(* PLC project Anjlab Code Box, Prosoft-Systems Ltd. Astra.IDE Astra.IDE_V1.7.2.1, author Sergey A Glukhov *)
(* stored: creationDateTime 2025-06-12T14:05:23.9971404, version 3.5.17.1, modificationDateTime 2025-06-12T13:59:54.8513333, organization Anjlab *)
(* Helpful ST blocks and functions *)

(* Сглаживание дискретного сигнала *)
FUNCTION_BLOCK DebunceBoolIn
  VAR_INPUT
    input : BOOL;  (* Входной сигнал *)
  END_VAR
  VAR_OUTPUT
    output : BOOL;  (* Выходной сигнал *)
  END_VAR
  VAR
    startTime : TIME;  (* Время начала *)
    memory : BOOL;  (* Память сигнала *)
  END_VAR

            IF input AND NOT memory THEN
	startTime := TIME();
END_IF;
memory := input;
output := input AND ((TIME() - startTime) > T#100ms);
          
END_FUNCTION_BLOCK

(* Сглаживание дискретного сигнала *)
FUNCTION_BLOCK DebunceBoolInOut
  VAR_INPUT
    input : BOOL;  (* Входной сигнал *)
  END_VAR
  VAR_OUTPUT
    output : BOOL;  (* Выходной сигнал *)
  END_VAR
  VAR
    startTime : TIME;  (* Время начала *)
    memory : BOOL;  (* Память сигнала *)
  END_VAR

            IF (NOT input AND memory) OR (input AND NOT memory) THEN
	startTime := TIME();
END_IF;
memory := input;
output := input;
IF ((TIME() - startTime) < T#100ms) THEN
	output := NOT input;
END_IF
          
END_FUNCTION_BLOCK

(* Сглаживание дискретного сигнала *)
FUNCTION_BLOCK DebunceBoolOut
  VAR_INPUT
    input : BOOL;  (* Входной сигнал *)
  END_VAR
  VAR_OUTPUT
    output : BOOL;  (* Выходной сигнал *)
  END_VAR
  VAR
    startTime : TIME;  (* Время начала *)
    memory : BOOL;  (* Память сигнала *)
  END_VAR

            IF NOT input AND memory THEN
	startTime := TIME();
END_IF;
memory := input;
output := input;
IF NOT input AND ((TIME() - startTime) < T#100ms) THEN
	output := TRUE;
END_IF
          
END_FUNCTION_BLOCK

(* выделяет передний и задний фронт с фильтром на 100 миллисекунд *)
FUNCTION_BLOCK DetectEdgeFiltered
  VAR_INPUT
    input : BOOL;  (* Входной сигнал *)
  END_VAR
  VAR_OUTPUT
    raise : BOOL;  (* Передний фронт *)
    fall : BOOL;  (* Задний фронт *)
  END_VAR
  VAR
    fbDio1 : DebunceBoolInOut;
    filteredInput : BOOL;  (* Отфильтрованный вход *)
    memory : BOOL;
  END_VAR

            fbDio1(input := input, output => filteredInput);
raise := fall := FALSE;
IF filteredInput AND NOT memory THEN
	raise := TRUE;
ELSIF NOT filteredInput AND memory THEN
	fall := TRUE;
END_IF
memory := filteredInput;
          
END_FUNCTION_BLOCK

(* Двойной клик *)
FUNCTION_BLOCK DoubleClick
  VAR_INPUT
    input : BOOL;  (* Входной сигнал *)
  END_VAR
  VAR_OUTPUT
    output : BOOL;  (* Выходной сигнал *)
  END_VAR
  VAR
    startTime : TIME;  (* Время начала *)
    memory : BOOL;  (* Память сигнала *)
  END_VAR

            output := FALSE;
IF input AND NOT memory THEN
	IF (TIME() - startTime) > T#100MS AND (TIME() - startTime) < T#800MS THEN
		output := TRUE;
	END_IF;
	startTime := TIME();
END_IF;
memory := input;
          
END_FUNCTION_BLOCK

(* Эта функция хранит до 32-х значений в буфере и выдает среднее значение. Вы сами можете решить, сколько значений сохранить для получения среднего числа. *)
FUNCTION_BLOCK FilterNR
  VAR_INPUT
    input : WORD;  (* Входное значение *)
    bufferSize : UINT;  (* Размер буфера минимум 32 максимум 1000 *)
    reset : BOOL;  (* Сброс буфера *)
  END_VAR
  VAR_OUTPUT
    output : WORD;  (* Выходное отфильтрованное значение *)
  END_VAR
  VAR
    isInitialized : BOOL;
    buffer : ARRAY[1..1000] OF WORD;
    counter : UINT;
    sum : DINT;
  END_VAR

            (* ограничим bufferSize в размер буфера *)
bufferSize := MIN(MAX(bufferSize, 1000), 32);
(* Инициализация *)
IF NOT isInitialized OR reset THEN
	isInitialized := TRUE;
	FOR counter := 1 TO bufferSize DO
		buffer[counter] := input;
	END_FOR;
	sum := input * bufferSize;
	output := input;
	RETURN;
END_IF;

IF counter >= bufferSize THEN
    counter := 1;
ELSE
    counter := counter + 1;
END_IF

sum := sum + input - buffer[counter];
{warning disable C0195}
output := DWORD_TO_WORD(sum / bufferSize);
buffer[counter] := input;
          
END_FUNCTION_BLOCK

(* возвращает среднее значение за определенный промежуток времени. *)
FUNCTION_BLOCK FilterTW
  VAR_INPUT
    input : WORD;  (* Входное значение *)
    timeInterval : TIME;  (* Временной интервал *)
  END_VAR
  VAR_OUTPUT
    output : WORD;  (* Выходное отфильтрованное значение *)
  END_VAR
  VAR
    isInitialized : BOOL;
    currentTime : DWORD;
    lastTime : DWORD;
    tempTime : DWORD;
  END_VAR

            (* Получаем текущее время *)
currentTime := TIME_TO_DWORD(TIME());
(* Инициализация *)
IF NOT isInitialized OR timeInterval = T#0s THEN
	isInitialized := TRUE;
	lastTime := currentTime;
	output := input;
ELSIF output = input THEN
	lastTime := currentTime;
ELSE
	tempTime := WORD_TO_DWORD(input - output) * (currentTime - lastTime) /
	TIME_TO_DWORD(timeInterval);
	IF tempTime <> 0 THEN
		output := DINT_TO_WORD(WORD_TO_DINT(output) + DWORD_TO_DINT(tempTime));
		lastTime := currentTime;
	END_IF;
END_IF;
          
END_FUNCTION_BLOCK

(* Долгий клик *)
FUNCTION_BLOCK LongClick
  VAR_INPUT
    input : BOOL;  (* Входной сигнал *)
    pressTime : TIME;  (* Время нажатия *)
  END_VAR
  VAR_OUTPUT
    output : BOOL;  (* Выходной сигнал *)
  END_VAR
  VAR
    startTime : TIME;  (* Время начала *)
    memory : BOOL;  (* Память сигнала *)
  END_VAR

            IF input AND NOT memory THEN
	startTime := TIME();
END_IF;
memory := input;
output := input AND ((TIME() - startTime) > pressTime);
          
END_FUNCTION_BLOCK

(* создает импульсы с заданной частотой CLK_PWM(EN := TRUE, PT := T#5ms); На выходе Q будет импульс в один цикл ПЛК, раз в 5 миллисекунд. *)
FUNCTION_BLOCK PwmClock
  VAR_INPUT
    enable : BOOL;  (* Запуск генератора *)
    pulseTime : TIME := TIME#10ms;  (* Время импульсов *)
  END_VAR
  VAR_OUTPUT
    output : BOOL;  (* Выходной сигнал *)
  END_VAR
  VAR
    memory : BOOL;
    lastTime : TIME;
    currentTime : TIME;
  END_VAR

            currentTime := TIME();
IF enable AND NOT memory THEN
	lastTime := currentTime - pulseTime;
END_IF;
memory := enable;
output := currentTime - lastTime >= pulseTime;
IF output THEN lastTime := currentTime; END_IF;
          
END_FUNCTION_BLOCK

(* создает ШИМ-сигнал заданной частоты со смещением соотношения. Каждый цик ШИМ можно разделить на 2 фазы: Ton (время включения) и Toff (время выключения). Соотношение задается от 0 до 1. Например, соотношение 0.5 разделит время каждого цикла шим на 50% на Ton и 50% на Toff . *)
FUNCTION_BLOCK PwmDc
  VAR_INPUT
    frequency : REAL;  (* Частота, раз в секунду (Гц) *)
    dutyCycle : REAL;  (* Соотношение *)
  END_VAR
  VAR_OUTPUT
    output : BOOL;  (* Выходной сигнал *)
  END_VAR
  VAR
    clock : PwmClock;
    pulseTimer : TP;
    tempValue : REAL;
  END_VAR

            (* Если частота ШИМ 0, то прерываем исполнение ФБ *)
IF frequency <= 0.0 THEN
	output := FALSE;
	RETURN;
END_IF;
(* Вычисляем сколько миллисекунд требуется на один цикл ШИМ *)
tempValue := 1000.0 / frequency;
(* Запускаем генератор сигналов *)
clock(pulseTime := REAL_TO_TIME(tempValue));
(* Создаем выдержанный пульс на нужное время *)
pulseTimer(in := clock.output, pt := REAL_TO_TIME(tempValue * dutyCycle), Q => output);
          
END_FUNCTION_BLOCK

(* Создает ШИМ-сигнал с заданным временем фазы Ton . Например, мы можем установить F на 100 раз в секунду. Это значит, один цикл ШИМ будет 10 миллисекунд. Теперь поставим PW в T#5ms и получим равное время для фазы Ton и Toff по 50%. *)
FUNCTION_BLOCK PwmPw
  VAR_INPUT
    frequency : REAL;  (* Частота, раз в секунду (Гц) *)
    pulseWidth : TIME;  (* Длина фазы Ton *)
  END_VAR
  VAR_OUTPUT
    output : BOOL;  (* Выходной сигнал *)
  END_VAR
  VAR
    clock : PwmClock;
    pulseTimer : TP;
  END_VAR

            (* Если частота ШИМ 0 или время одного цикла меньше,
чем время для фазы Ton, то прерываем исполнение ФБ *)
IF frequency <= 0.0 OR (REAL_TO_TIME(1000.0 / frequency) < pulseWidth) THEN
	output := FALSE;
	RETURN;
END_IF;
(* Запускаем генератор сигналов *)
clock(pulseTime := REAL_TO_TIME(1000.0 / frequency));
(* Создаем выдержанный пульс на нужное время *)
pulseTimer(in := clock.output, PT := pulseWidth, Q => output);
          
END_FUNCTION_BLOCK

(* расчет времени заката и восхода *)
FUNCTION_BLOCK SunTime
  VAR_INPUT
    LATITUDE : REAL;  (* Широта *)
    LONGITUDE : REAL;  (* Долгота *)
    UTC : DATE;  (* Текущее время в UTC *)
    H : REAL := -0.83333333333;  (* Градус над горизонтом, при котором уже считается наступление заката или восхода *)
  END_VAR
  VAR_OUTPUT
    MIDDAY : TOD;  (* Время дня солнцестояния *)
    SUN_RISE : TOD;  (* Время восхода *)
    SUN_SET : TOD;  (* Время заката *)
    SUN_DECLINATION : REAL;  (* Угол наклона солнца в солнцестояние в градусах *)
  END_VAR
  VAR
    dk : REAL;  (* Угол наклона солнца в полдень в радианах *)
    delta : TIME;  (* Дельта от солнцестояния до восхода или заката *)
    b : REAL;
  END_VAR

            MIDDAY := SunMidday(longitude, utc);
b := latitude * 0.0174532925199433;
dk := 0.40954 * SIN(0.0172 * (UINT_TO_REAL(DayOfYear(utc)) - 79.35));
SUN_DECLINATION := DegreesToRadians(DK);
IF SUN_DECLINATION > 180.0 THEN
	SUN_DECLINATION := SUN_DECLINATION - 360.0;
END_IF;
SUN_DECLINATION := 90.0 - LATITUDE + SUN_DECLINATION;
delta := HourToTime(REAL_TO_INT(ACOS((SIN(RadiansToDegrees(H)) - SIN(B) * SIN(DK)) / (COS(B) * COS(DK))) * 3.819718632));
SUN_RISE := MIDDAY - delta;
SUN_SET := MIDDAY + delta;
          
END_FUNCTION_BLOCK

(* Преобразование в шестнадцатеричный формат для записи IP *)
FUNCTION IpDecode : DWORD
  VAR_INPUT
    ipStr : STRING(15);  (* IP-адрес как строка, например, '192.168.1.2' *)
  END_VAR
  VAR
    position : INT;
  END_VAR

            position := FIND(ipStr, '.');
WHILE position > 0 DO
	IpDecode := SHL(IpDecode, 8) OR
	STRING_TO_DWORD(LEFT(ipStr, position - 1));
	ipStr := DELETE(ipStr, position, 1);
	position := FIND(ipStr, '.');
END_WHILE;
IpDecode := SHL(IpDecode, 8) OR STRING_TO_DWORD(ipStr);
          
END_FUNCTION

(* Округляет значение и возвращает ближайшее целое значение, которое больше или равно X. ceil(3.14) = 4 ceil(-3.14) = -3 *)
FUNCTION Ceil : DINT
  VAR_INPUT
    input : REAL;  (* Входное значение *)
  END_VAR

            Ceil := REAL_TO_DINT(input);

IF DINT_TO_REAL(Ceil) < input THEN
	Ceil := Ceil + 1;
END_IF;
          
END_FUNCTION

(* Вычисляет с основанием степени 10. exp10(2) = 100 exp10(3) = 1000 *)
FUNCTION Exp10 : REAL
  VAR_INPUT
    input : REAL;  (* Входное значение *)
  END_VAR

            Exp10 := EXP(input * 2.30258509299405);
          
END_FUNCTION

(* Возведение в степень X^N. Хотя в стандарте есть оператор EXPT, по заявлению OSCAT, данный алгоритм работает в 30 раз быстрее в CoDeSys. *)
FUNCTION ExpN : REAL
  VAR_INPUT
    input : REAL;  (* Входное значение *)
    power : INT;  (* Степень *)
  END_VAR
  VAR
    sign : BOOL;
  END_VAR

            sign := power.15;
power := ABS(power);
IF power.0 THEN ExpN := input; ELSE ExpN := 1.0; END_IF;
power := SHR(power, 1);

WHILE power > 0 DO
	input := input * input;
	IF power.0 THEN ExpN := ExpN * input; END_IF;
	power := SHR(power, 1);
END_WHILE;

IF sign THEN ExpN := 1.0 / ExpN; END_IF;
          
END_FUNCTION

(* Округляет значение и возвращает ближайшее целое значение, которое меньше или равно X. floor(3.14) = 3 floor(-3.14) = -4 *)
FUNCTION Floor : DINT
  VAR_INPUT
    input : REAL;  (* Входное значение *)
  END_VAR

            FLOOR := REAL_TO_DINT(input);
IF DINT_TO_REAL(FLOOR) > input THEN
	FLOOR := FLOOR - 1;
END_IF;
          
END_FUNCTION

(* Эта функция возвращает дробную часть числа с плавающей точкой. fract(3.14) = 0.14 *)
FUNCTION Fract : REAL
  VAR_INPUT
    input : REAL;  (* Входное значение *)
  END_VAR

            IF ABS(input) < 2.0E9 THEN
	FRACT := input - DINT_TO_REAL(DTrunc(input));
ELSE
	FRACT := 0.0;
END_IF;
          
END_FUNCTION

(* Вычисляет остаток от деления для чисел с плавающей запятой. modr(5.5, 2.5) = 0.5 *)
FUNCTION ModR : REAL
  VAR_INPUT
    input : REAL;  (* Делимое *)
    divisor : REAL;  (* Делитель *)
  END_VAR

            IF divisor = 0.0 THEN
	MODR := 0.0;
ELSE
	MODR := input - DINT_TO_REAL(FLOOR(input / divisor)) * divisor;
END_IF;

          
END_FUNCTION

(* Округляет число с плавающей точкой до указанного количества знаков после запятой. round(12.23456789, 2) = 12.23 *)
FUNCTION Round : REAL
  VAR_INPUT
    input : REAL;  (* Число для обработки *)
    precision : USINT;  (* Точность после запятой *)
  END_VAR

            Round := DWORD_TO_REAL(REAL_TO_DWORD(input * Exp10(precision))) / Exp10(precision);

          
END_FUNCTION

(* Преобразование температуры из Цельсия в Фаренгейт *)
FUNCTION CelciusToFarenheit : REAL
  VAR_INPUT
    celsiusTemp : REAL;  (* Входное значение в Цельсиях *)
  END_VAR

            CelciusToFarenheit := celsiusTemp * 1.8 + 32.0;
          
END_FUNCTION

(* Преобразование температуры из Цельсия в Кельвин *)
FUNCTION CelciusToKelvin : REAL
  VAR_INPUT
    celsiusTemp : REAL;  (* Входное значение в Цельсиях *)
  END_VAR
  VAR CONSTANT
    physT0 : REAL := 273.15;  (* 0°C в кельвинах *)
  END_VAR

            CelciusToKelvin := celsiusTemp + physT0;
          
END_FUNCTION

(* Конвертирует радианы в градусы. *)
FUNCTION DegreesToRadians : REAL
  VAR_INPUT
    radians : REAL;  (* Входное значение в радианах *)
  END_VAR

            DegreesToRadians := ModR(57.29577951308232 * radians, 360.0);
          
END_FUNCTION

(* Преобразование температуры из Фаренгейт в Цельсий *)
FUNCTION FarenheitToCelcius : REAL
  VAR_INPUT
    fahrenheitTemp : REAL;  (* Входное значение в Фаренгейтах *)
  END_VAR

            FarenheitToCelcius := (fahrenheitTemp - 32.0) * 0.5555555555555;
          
END_FUNCTION

(* Преобразование температуры из Кельвина в Цельсий *)
FUNCTION KelvinToCelcius : REAL
  VAR_INPUT
    kelvinTemp : REAL;  (* Входное значение в Кельвнах *)
  END_VAR
  VAR CONSTANT
    phys_T0 : REAL := 273.15;  (* 0°C в кельвинах *)
  END_VAR

            KelvinToCelcius := kelvinTemp - phys_T0;
          
END_FUNCTION

(* Преобразование скорости: км/ч в м/с *)
FUNCTION KmhToMs : REAL
  VAR_INPUT
    kmhSpeed : REAL;  (* Входное значение в Км/ч *)
  END_VAR

            KmhToMs := kmhSpeed * 0.2777777777777;
          
END_FUNCTION

(* Преобразование скорости: м/с в км/ч *)
FUNCTION MsToKmh : REAL
  VAR_INPUT
    msSpeed : REAL;  (* Входное значение в м/с *)
  END_VAR

            MsToKmh := msSpeed * 3.6;
          
END_FUNCTION

(* конвертирует градусы в радианы *)
FUNCTION RadiansToDegrees : REAL
  VAR_INPUT
    degrees : REAL;  (* Входное значение в градусах *)
  END_VAR
  VAR
    timeNow : DWORD;
    timeCount : INT;
  END_VAR
  VAR CONSTANT
    pi : REAL := 3.1415926535897931;
  END_VAR

            RadiansToDegrees := ModR(0.0174532925199433 * degrees, pi*2);
          
END_FUNCTION

(* линейное масштабирование числа с плавающей запятой *)
FUNCTION ScaleReal : REAL
  VAR_INPUT
    input : REAL;  (* Входное значение *)
    inputLow : REAL;  (* Входное минимальное *)
    inputHigh : REAL;  (* Входное максимальное *)
    outputLow : REAL;  (* Выходное минимальное *)
    outputHigh : REAL;  (* Выходное максимальное *)
  END_VAR

            IF inputLow = inputHigh THEN
	ScaleReal := outputLow;
ELSE
	ScaleReal := (outputHigh - outputLow) / (inputHigh - inputLow) * (LIMIT(inputLow, input, inputHigh) - inputLow) + outputLow;
END_IF;
          
END_FUNCTION

(* считает, как много указанных символов содержится в строке *)
FUNCTION CountChar : INT
  VAR_INPUT
    inputString : STRING(255);  (* Строка *)
    charToCount : BYTE;  (* Символ для подсчета *)
  END_VAR
  VAR
    charPointer : POINTER TO BYTE;  (* Указатель на символ *)
    length : INT;  (* Длина строки *)
    position : INT;  (* Текущая позиция строки для прохода *)
  END_VAR

            charPointer := ADR(inputString);
length := LEN(inputString);
CountChar := 0;
FOR position := 1 TO length DO
	IF charPointer^ = charToCount THEN
		CountChar := CountChar + 1;
	END_IF;
	charPointer := charPointer + 1;
END_FOR;
          
END_FUNCTION

(* Удаление символа из строки *)
FUNCTION RemoveSubString : STRING
  VAR_INPUT
    inputString : STRING;  (* Входная строка *)
    substringToRemove : STRING;  (* Что удалить *)
  END_VAR
  VAR
    tempString : STRING;  (* Для временной строки *)
    position : INT;  (* Позиция найденного символа *)
  END_VAR

            tempString := inputString;
REPEAT
	position := FIND(tempString, substringToRemove);
	IF position <> 0 THEN
		tempString := DELETE(tempString, LEN(substringToRemove), position);
	END_IF;
UNTIL (position = 0)
END_REPEAT;
RemoveSubString := tempString;
          
END_FUNCTION

(* Изменить регистр символа с маленькой буквы на заглавную. Работает только с латинскими буквами формата ASCII. *)
FUNCTION ToUpper : BYTE
  VAR_INPUT
    input : BYTE;  (* Входная строка *)
    useExtendedASCII : BOOL;  (* Значение setup.EXTENDED_ASCII может быть или TRUE или FALSE, в зависимости от символьной таблицы, которая поддерживается ПЛК. Обычно стоит в TRUE. *)
  END_VAR

            IF input > 96 AND input < 123 THEN
	ToUpper := input AND 16#DF;
ELSIF input > 223 AND input <> 247 AND input <> 255 AND useExtendedASCII THEN
	ToUpper := input AND 16#DF;
ELSE
	ToUpper := input;
END_IF;
          
END_FUNCTION

(* Извлечение года, месяца и дня из DATE *)
FUNCTION DateToElements : BOOL
  VAR_INPUT
    input : DATE;  (* Входная дата *)
  END_VAR
  VAR_OUTPUT
    year : UINT;  (* Год *)
    month : UINT;  (* Месяц *)
    day : UINT;  (* День *)
  END_VAR
  VAR
    sTemp : STRING;
  END_VAR

            (* Получаем дату строкой 'D#2000-01-01' *)
sTemp := DATE_TO_STRING(input);
year := STRING_TO_UINT(MID(sTemp, 3, 4));
month := STRING_TO_UINT(MID(sTemp, 8, 2));
day := STRING_TO_UINT(MID(sTemp, 11, 2));

DateToElements := true;
          
END_FUNCTION

(* Определение дня недели *)
FUNCTION DayOfWeek : UINT
  VAR_INPUT
    input : DATE;  (* Входная дата *)
  END_VAR
  VAR
    NumOfDay : DWORD;
  END_VAR

            NumOfDay := DATE_TO_DWORD(input) / 86400; 
NumOfDay := NumOfDay + 3;
DayOfWeek := DWORD_TO_UINT(NumOfDay MOD 7);
          
END_FUNCTION

(* Вычисление порядкового дня в году *)
FUNCTION DayOfYear : UINT
  VAR_INPUT
    input : DATE;  (* Входная дата в формате DATE *)
  END_VAR
  VAR
    year : UINT;
    month : UINT;
    day : UINT;
  END_VAR

            DateToElements(input := input, year => year, month => month, day => day);

DayOfYear := DaysTillMonth(year, month) + day;
          
END_FUNCTION

(* Вычисление количества дней в году *)
FUNCTION DaysInYear : UINT
  VAR_INPUT
    year : UINT;  (* Год *)
  END_VAR

            IF IsLeapYear(year) THEN
	DaysInYear := 366;
ELSE
	DaysInYear := 365;
END_IF;
          
END_FUNCTION

(* функция, чтобы определить количество дней от начала года до указанного месяца. *)
FUNCTION DaysTillMonth : UINT
  VAR_INPUT
    year : UINT;  (* Год *)
    month : UINT;  (* Месяц *)
  END_VAR
  VAR
    days : ARRAY[1..12] OF UINT := [0, 31, 59, 90, 120, 151, 181, 212, 243, 273, 304, 334];
  END_VAR

            DaysTillMonth := days[month] + BOOL_TO_UINT(month > 2 AND IsLeapYear(year));
          
END_FUNCTION

(* считает сколько прошло дней до указанного года *)
FUNCTION DaysTillYear : UINT
  VAR_INPUT
    year : UINT;  (* Год *)
  END_VAR

            (* Получаем количество лет прошло с 1970го года *)
year := year - 1970;
DaysTillYear := year * 365 + ((year + 1) / 4) - ((year + 69) / 100) + ((year + 369) / 400);
          
END_FUNCTION

(* Упаковка часов, минут, секунд и миллисекунд в TIME *)
FUNCTION HmsToTime : TIME
  VAR_INPUT
    h : UINT;  (* Часы *)
    m : UINT;  (* Минуты *)
    sec : UINT;  (* Секунды *)
    ms : UINT;  (* Миллисекунды *)
  END_VAR

            HmsToTime := DWORD_TO_TIME(((h * 60 + m) * 60 + sec) * 1000 + ms);
          
END_FUNCTION

(* Преобразовать часы (в виде INT) в TIME *)
FUNCTION HourToTime : TIME
  VAR_INPUT
    hours : INT;  (* Часы (0..23) *)
  END_VAR

            HourToTime := T#1H * hours;
          
END_FUNCTION

(* Преобразовать количество часов (INT) во значение типа TOD (время суток). *)
FUNCTION HourToTod : TOD
  VAR_INPUT
    hours : INT;  (* Часы (0..23) *)
  END_VAR

            HourToTod := TOD#00:00:00 + T#1h * hours;
          
END_FUNCTION

(* Определение високосного года *)
FUNCTION IsLeapYear : BOOL
  VAR_INPUT
    year : UINT;  (* Год *)
  END_VAR

            IsLeapYear := year MOD 400 = 0 OR year MOD 4 = 0 AND year MOD 100 <> 0;
          
END_FUNCTION

(* время солнцестояния на заданной широте в заданное время *)
FUNCTION SunMidday : TOD
  VAR_INPUT
    LON : REAL;  (* Широта *)
    UTC : DATE;  (* Дата в UTC *)
  END_VAR
  VAR
    T : REAL;
    OFFSET : REAL;
  END_VAR

            T := UINT_TO_REAL(DayOfYear(utc));
OFFSET := -0.1752 * SIN(0.033430 * T + 0.5474) - 0.1340 * SIN(0.018234 * T - 0.1939);
SunMidday := HourToTod(REAL_TO_INT(12.0 - OFFSET - lon * 0.0666666666666));
          
END_FUNCTION

(* Извлечение часов, минут, секунд и миллисекунд из TIME *)
FUNCTION TimeToElements : BOOL
  VAR_INPUT
    input : TIME;  (* Входное время *)
  END_VAR
  VAR_OUTPUT
    h : UINT;
    m : UINT;
    sec : UINT;
    ms : UINT;
  END_VAR
  VAR
    sTemp : STRING;
  END_VAR

            (* Теперь время имеет строку типа 'TOD#12:12:59' *)
sTemp := TOD_TO_STRING(TIME_TO_TOD(input));
h := STRING_TO_UINT(MID(sTemp, 5, 2));
m := STRING_TO_UINT(MID(sTemp, 8, 2));
sec := STRING_TO_UINT(MID(sTemp, 11, 2));
TimeToElements := TRUE;
          
END_FUNCTION

(* функция определения, что текущее время находится в промежутке между двумя отметками времени TIME_OF_DAY. *)
FUNCTION TodBetween : BOOL
  VAR_INPUT
    CurrTime : TOD;  (* текущее время *)
    FromTime : TOD;  (* нижняя граница *)
    ToTime : TOD;  (* верхняя граница *)
  END_VAR

            TodBetween := (
	FromTime > ToTime AND (CurrTime > FromTime OR CurrTime < ToTime)
	) OR (FromTime < ToTime AND (CurrTime < ToTime AND CurrTime > FromTime)
);

          
END_FUNCTION

(* Вычисление разницы отметок времени *)
FUNCTION TodDiff : TIME
  VAR_INPUT
    FromTime : TOD;  (* нижняя граница *)
    ToTime : TOD;  (* верхняя граница *)
  END_VAR

            IF ToTime < FromTime THEN
	TodDiff := T#24H - TOD_TO_TIME(FromTime) + TOD_TO_TIME(ToTime);
ELSE
	TodDiff := ToTime - FromTime;
END_IF
          
END_FUNCTION

(* Вычисления порядкового номера недели в году *)
FUNCTION WeekOfYear : UINT
  VAR_INPUT
    currentDate : DATE;  (* Текущая дата *)
  END_VAR

            WeekOfYear := ((DayOfYear(currentDate) + 6) / 7);
IF DayOfWeek(currentDate) < DayOfWeek(YearStarts(currentDate)) THEN
	WeekOfYear := WeekOfYear + 1;
END_IF;
          
END_FUNCTION

(* Вычисления с какого дня недели начинается год *)
FUNCTION YearStarts : DATE
  VAR_INPUT
    currentDate : DATE;  (* Текущая дата *)
  END_VAR
  VAR
    str : STRING(25);  (* Временная строка *)
  END_VAR

            str := DATE_TO_STRING(currentDate); (* получаем строку `D#2000-12-30` *)
YearStarts := STRING_TO_DATE(CONCAT(CONCAT('D#', MID(str, 3, 4)), '-01-01'));
          
END_FUNCTION

(* Упаковка года, месяца, дня, часов, минут, секунд и миллисекунд в DT *)
FUNCTION YmdhmsTodt : DT
  VAR_INPUT
    y : UINT;  (* Год *)
    mn : UINT;  (* Месяц *)
    d : UINT;  (* День *)
    h : UINT;  (* Час *)
    m : UINT;  (* Минуты *)
    sec : UINT;  (* Секунды *)
    ms : UINT;  (* Миллисекунды *)
  END_VAR
  VAR
    sTemp : STRING;
  END_VAR

            sTemp := CONCAT('DT#', UINT_TO_STRING(y));
sTemp := CONCAT(sTemp, '-');
sTemp := CONCAT(sTemp, UINT_TO_STRING(mn));
sTemp := CONCAT(sTemp, '-');
sTemp := CONCAT(sTemp, UINT_TO_STRING(d));
sTemp := CONCAT(sTemp, '-');
sTemp := CONCAT(sTemp, UINT_TO_STRING(h));
sTemp := CONCAT(sTemp, '-');
sTemp := CONCAT(sTemp, UINT_TO_STRING(m));
sTemp := CONCAT(sTemp, '-');
sTemp := CONCAT(sTemp, UINT_TO_STRING(sec));
sTemp := CONCAT(sTemp, '-');
sTemp := CONCAT(sTemp, UINT_TO_STRING(ms));
YmdhmsTodt := STRING_TO_DT(sTemp);
          
END_FUNCTION

(* Gеревод год, месяц и день в формат DATE. *)
FUNCTION YmdToDate : DATE
  VAR_INPUT
    y : UINT;  (* Год *)
    m : UINT;  (* Месяц *)
    d : UINT;  (* День *)
  END_VAR
  VAR
    sTemp : STRING;
  END_VAR

            sTemp := CONCAT('D#', UINT_TO_STRING(y));
sTemp := CONCAT(sTemp, '-');
sTemp := CONCAT(sTemp, UINT_TO_STRING(m));
sTemp := CONCAT(sTemp, '-');
sTemp := CONCAT(sTemp, UINT_TO_STRING(d));
YmdToDate := STRING_TO_DATE(sTemp);
          
END_FUNCTION

(* Cчитает количество бит, равных TRUE в DWORD. Пример: bit_count(3) = 2 Потому что 2 бита равны 1, а остальные равны 0. *)
FUNCTION BitCount : INT
  VAR_INPUT
    input : DWORD;  (* Входное число *)
  END_VAR

            WHILE input > 0 DO
	IF input.0 THEN
		BitCount := BitCount + 1;
	END_IF
	input := SHR(input, 1);
END_WHILE;
          
END_FUNCTION

(* Загружает значение одного бита в байт. bit_load_b(2#0000_0000, 1, 2) = 2#0000_0010 *)
FUNCTION BitLoadB : BYTE
  VAR_INPUT
    input : BYTE;  (* Байт, в котором нужно произвести операцию *)
    value : BOOL;  (* Присваиваемое значение *)
    position : INT;  (* Какому по номеру биту *)
  END_VAR
  VAR CONSTANT
    dat : BYTE := 1;
  END_VAR

            IF value THEN
	BitLoadB := input OR SHL(dat, position);
ELSE
	BitLoadB := input AND (NOT SHL(dat, position));
END_IF;
          
END_FUNCTION

(* Вычисляем значение единичного бита в переменной типа DWORD. *)
FUNCTION BitOfDword : BOOL
  VAR_INPUT
    input : DWORD;  (* Входное число *)
    n : INT;  (* номер бита *)
  END_VAR

            BitOfDword := (SHR(input, n) AND 16#00000001) > 0;
          
END_FUNCTION

(* Инвертируем указанный бит в DWORD *)
FUNCTION BitToggleDword : DWORD
  VAR_INPUT
    input : DWORD;  (* Входное значение *)
    position : INT;  (* Номер инвертируемого бита *)
  END_VAR

            BitToggleDword := SHL(DWORD#1, position) XOR input;
          
END_FUNCTION

(* Сравнивает 2 входных числовых переменных, совпадают ли их первые разрады. Количество сравниваемых разрядов передается в параметре N. cmp(3.141516, 3.141517, 6) вернет TRUE. *)
FUNCTION CompareReals : BOOL
  VAR_INPUT
    x : REAL;  (* Входное значение X *)
    y : REAL;  (* Входное значение Y *)
    n : INT;  (* Количество сравниваемых разрядов *)
  END_VAR
  VAR
    tmp : REAL;
  END_VAR

            tmp := ABS(x);
IF tmp > 0.0 THEN
	tmp := Exp10(DINT_TO_REAL(FLOOR(LOG(tmp))-n+1));
ELSE
	tmp := Exp10(tmp);
END_IF;

CompareReals := ABS(x - y) < tmp;
          
END_FUNCTION

(* Усекает число с плавающей запятой в целое число DINT. 1.5 станет 1, а -1.5 станет -1. Данная функция необходима, потому что REAL_TO_DINT на разных системах может вернуть разный результат. *)
FUNCTION DTrunc : DINT
  VAR_INPUT
    input : REAL;  (* Входное значение *)
  END_VAR

            DTrunc := REAL_TO_DINT(input);

IF input > 0.0 THEN
	IF DINT_TO_REAL(DTrunc) > input THEN
		DTrunc := DTrunc - 1;
	END_IF;
ELSE
	IF DINT_TO_REAL(DTrunc) < input THEN
		DTrunc := DTrunc + 1;
	END_IF;
END_IF;
          
END_FUNCTION

(* Вычисляет, является ли число четным или нет. Если четное, то вернет TRUE, а если нет - вернет FALSE. *)
FUNCTION Even : BOOL
  VAR_INPUT
    input : DINT;  (* Входное значение *)
  END_VAR

            Even := NOT input.0;
          
END_FUNCTION

(* Вычисляет псевдо-случайное число. Чтобы сгенерировать число, функция считывает таймер ПЛК и создает число с плавающей точкой от 0 до 1. Чтобы использовать эту функцию больше, чем один раз, в одном цикле ПЛК, нужно ее вызывать с разным значением входного параметра last. В него проще внести прошлое число, чтобы исключить повторения. *)
FUNCTION Random : REAL
  VAR_INPUT
    last : REAL;  (* Предыдущее значение *)
  END_VAR
  VAR
    tn : DWORD;
    tc : INT;
  END_VAR
  VAR CONSTANT
    E : REAL := 2.7182818284590451;  (* константа Эйлера *)
  END_VAR

            tn := TIME_TO_DWORD(TIME());
tc := BitCount(tn);
tn.31 := tn.2;
tn.30 := tn.5;
tn.29 := tn.4;
tn.28 := tn.1;
tn.27 := tn.0;
tn.26 := tn.7;
tn.25 := tn.6;
tn.24 := tn.3;
tn := ROL(tn, BitCount(tn)) OR 16#80000001;
tn := tn MOD 71474513 + INT_TO_DWORD(tc + 77);
Random := FRACT(DWORD_TO_REAL(tn) / 10000000.0 *
(E - LIMIT(0.0, last, 1.0))
);
          
END_FUNCTION

(* Поменять байт местами в DWORD *)
FUNCTION SwapDwordBytes : DWORD
  VAR_INPUT
    input : DWORD;  (* Входное значение *)
  END_VAR

            SwapDwordBytes := (ROR(input, 8) AND 16#FF00FF00) OR (ROL(input, 8) AND 16#00FF00FF);
          
END_FUNCTION

(* Поменять байт местами в WORD *)
FUNCTION SwapWordBytes : WORD
  VAR_INPUT
    input : WORD;  (* Входное значение *)
  END_VAR

            SwapWordBytes := ROL(input, 8);
          
END_FUNCTION
